INTERFACE I_Task EXTENDS __SYSTEM.IQueryInterface

METHOD Abort : BOOL
VAR_INPUT
END_VAR
END_METHOD

PROPERTY Busy : bool
GET
END_GET
END_PROPERTY

PROPERTY Done : bool
GET
END_GET
END_PROPERTY

PROPERTY Error : bool
GET
END_GET
END_PROPERTY

END_INTERFACE

(* stored: Version 1.1.0.1
   Itf I_Task: Id {d5273dc3-25ad-4a63-8b13-a40daf64efb7}
   Method Abort: Id {85cf1727-773a-4df7-85ee-41d8de64a86a}
   Property Busy: Id {b69f3fa5-0fc5-443d-ba3d-6e3f7de8be82}
   Get Get: Id {c4f84218-6027-49b0-a856-3fa8eac66e0a}
   Property Done: Id {edce6289-f58d-422a-93ec-31509bbce57e}
   Get Get: Id {3258da58-9596-4d92-9fc6-e49caff242bc}
   Property Error: Id {a2d0feb2-c8d3-4acc-84d1-e4f324066775}
   Get Get: Id {1ff60d1a-9bd0-4dc9-b0cf-6581a117847c} *)
